(* Logix 5000 project; controller TBEN_Lx_8IOL_AOI_V0_1 vendor 1 type 14 code 176 rev 32.11; software revision 32.00; part 11 of 11 *)
(* tags used below, declared in another part *)
   Port : INT;
   Universal_IOLink_Info : Universal_IOLink_Info;
   StartupDone : BOOL;
   Done : DINT;
   Error : DINT;
   Active : DINT;
   Pending : DINT;
   Pending_or_Active : DINT;
   Status : DINT;
   ErrorCount : DINT;
   Prev_Vendor_ID : INT;
(* Universal_Device_Info, continued *)

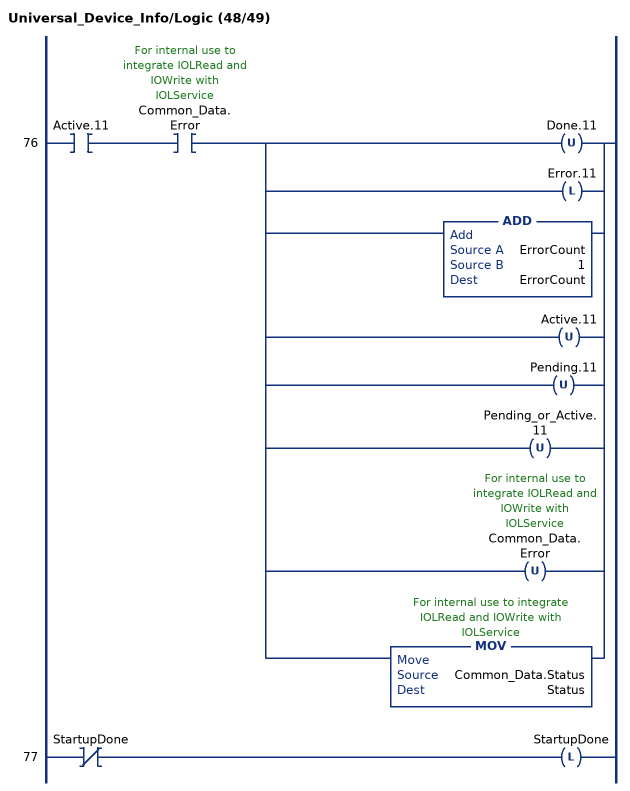
   [picture p96: Universal_Device_Info/Logic rungs 76-77]
   76: XIC(Active.11)XIC(Common_Data.Error)[OTU(Done.11) ,OTL(Error.11) ,ADD(ErrorCount,1,ErrorCount) ,OTU(Active.11) ,OTU(Pending.11) ,OTU(Pending_or_Active.11) ,OTU(Common_Data.Error) ,MOV(Common_Data.Status,Status) ];
   77: XIO(StartupDone)OTL(StartupDone);
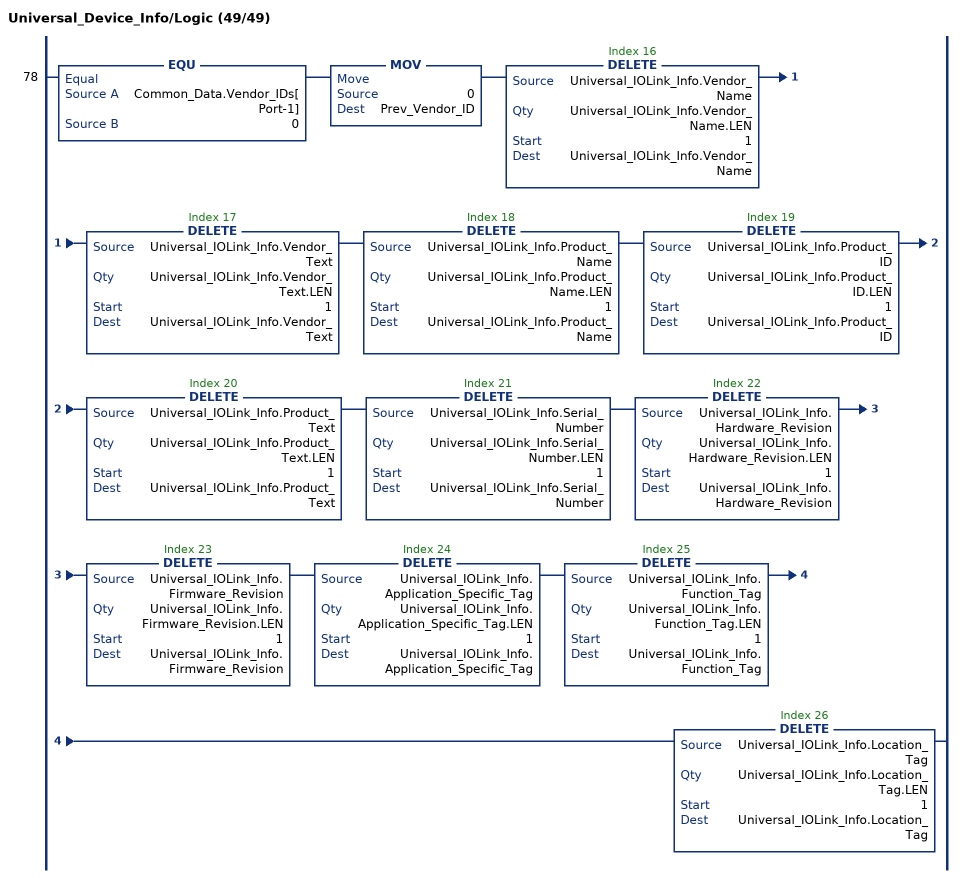
   78: EQU(Common_Data.Vendor_IDs[Port-1],0)MOV(0,Prev_Vendor_ID)DELETE(Universal_IOLink_Info.Vendor_Name,Universal_IOLink_Info.Vendor_Name.LEN,1,Universal_IOLink_Info.Vendor_Name)DELETE(Universal_IOLink_Info.Vendor_Text,Universal_IOLink_Info.Vendor_Text.LEN,1,Universal_IOLink_Info.Vendor_Text)DELETE(Universal_IOLink_Info.Product_Name,Universal_IOLink_Info.Product_Name.LEN,1,Universal_IOLink_Info.Product_Name)DELETE(Universal_IOLink_Info.Product_ID,Universal_IOLink_Info.Product_ID.LEN,1,Universal_IOLink_Info.Product_ID)DELETE(Universal_IOLink_Info.Product_Text,Universal_IOLink_Info.Product_Text.LEN,1,Universal_IOLink_Info.Product_Text)DELETE(Universal_IOLink_Info.Serial_Number,Universal_IOLink_Info.Serial_Number.LEN,1,Universal_IOLink_Info.Serial_Number)DELETE(Universal_IOLink_Info.Hardware_Revision,Universal_IOLink_Info.Hardware_Revision.LEN,1,Universal_IOLink_Info.Hardware_Revision)DELETE(Universal_IOLink_Info.Firmware_Revision,Universal_IOLink_Info.Firmware_Revision.LEN,1,Universal_IOLink_Info.Firmware_Revision)DELETE(Universal_IOLink_Info.Application_Specific_Tag,Universal_IOLink_Info.Application_Specific_Tag.LEN,1,Universal_IOLink_Info.Application_Specific_Tag)DELETE(Universal_IOLink_Info.Function_Tag,Universal_IOLink_Info.Function_Tag.LEN,1,Universal_IOLink_Info.Function_Tag)DELETE(Universal_IOLink_Info.Location_Tag,Universal_IOLink_Info.Location_Tag.LEN,1,Universal_IOLink_Info.Location_Tag);
END_ROUTINE

ROUTINE Prescan   (* ladder *)
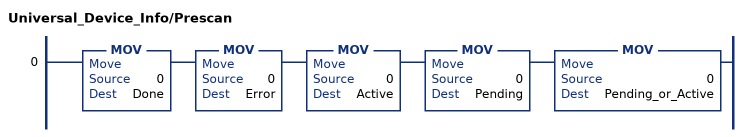
   0: MOV(0,Done)MOV(0,Error)MOV(0,Active)MOV(0,Pending)MOV(0,Pending_or_Active);
END_ROUTINE
END_ADD_ON_INSTRUCTION

VAR_GLOBAL   (* controller tags *)
   Common_Data : Turck_IOLink_Common_Data := (Port := 128, Index := -1, SubIndex := 68, Length := 224, NextTicketNum := 1, Process_Input_Data[0] := 192, ReceiveData[10] := 1, ReceiveData[11] := 61, ReceiveData[13] := 30, ReceiveData[14] := 51, ReceiveData[15] := 3, ReceiveData[18] := 48, ReceiveData[19] := 48, ReceiveData[20] := 48, ReceiveData[21] := 49, ReceiveData[22] := 48, ReceiveData[23] := 55, ReceiveData[24] := 54, ReceiveData[25] := 54, ReceiveData[26] := 53, ReceiveData[27] := 56, ReceiveData[28] := 45, ReceiveData[29] := 48, ReceiveData[30] := 48, ReceiveData[31] := 48, ReceiveData[32] := 50, ReceiveData[33] := 48, ReceiveData[34] := 17, ReceiveData[35] := 16, ReceiveData[36] := 16, ReceiveData[37] := 32, SendData[0] := -1, SendData[1] := -1, SendData[2] := 68, Vendor_IDs[0] := 317, Device_IDs[0] := 1979139);
   IOL_READ_MSG : MESSAGE;
        MessageParameters(ServiceCode := 16#004b, LocalElement := Common_Data.SendData, DestinationTag := Common_Data.ReceiveData, ...)
   IOL_WRITE_MSG : MESSAGE;
        MessageParameters(ServiceCode := 16#004c, LocalElement := Common_Data.SendData, DestinationTag := Common_Data.ReceiveData, ...)
   TBEN_8IOL_101 : TBEN_Lx_8IOL_AOI;
   TBEN_8IOL_101_Config_Tags_IN : Generic_160_SINT;
   TBEN_8IOL_101_Config_Tags_OUT : Generic_160_SINT;
   TBEN_8IOL_101_Process_Data_In : Generic_173_Words := (Data[0] := 1, Data[2] := 1, Data[3] := 192, Data[134] := 4, Data[135] := 4, Data[136] := 4, Data[137] := 4, Data[138] := 4, Data[139] := 4, Data[140] := 4);
   TBEN_8IOL_101_Process_Data_Out : Generic_131_Words;
   TBIL : Universal_Device_Info := (Port := 5);
   TBIL_Info : Universal_IOLink_Info;
   TEST : BOOL;
END_VAR

PROGRAM MainProgram   (* main routine MainRoutine *)
VAR
   TBEN_8IOL_100_Process_Data_In : Generic_173_Words := (Data[0] := 1, Data[133] := 4, Data[134] := 4, Data[135] := 4, Data[136] := 4, Data[137] := 4, Data[138] := 4, Data[139] := 4, Data[140] := 4);
   TBEN_8IOL_100_Process_Data_Out : Generic_131_Words;
END_VAR

ROUTINE MainRoutine   (* ladder *)
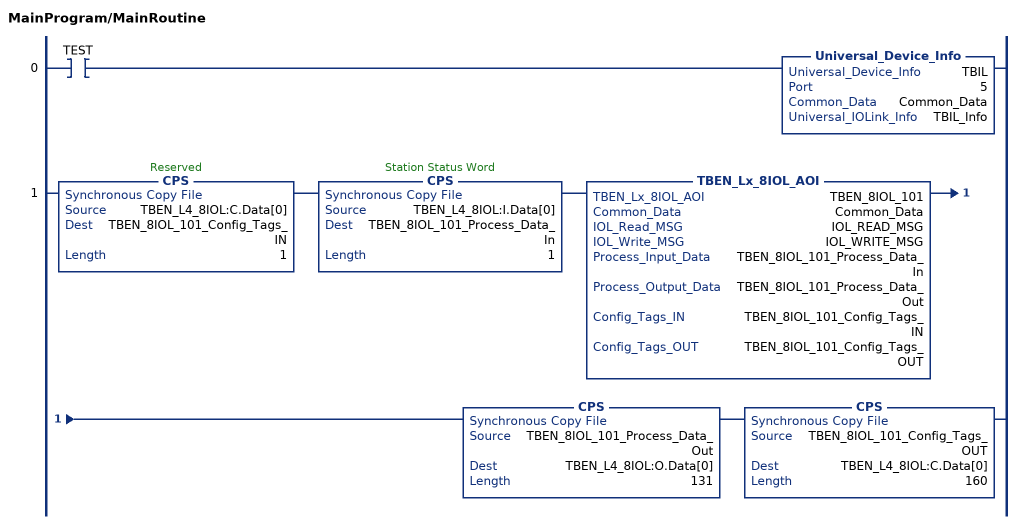
   0: XIC(TEST)Universal_Device_Info(TBIL,5,Common_Data,TBIL_Info);
   1: CPS(TBEN_L4_8IOL:C.Data[0],TBEN_8IOL_101_Config_Tags_IN,1)CPS(TBEN_L4_8IOL:I.Data[0],TBEN_8IOL_101_Process_Data_In,1)TBEN_Lx_8IOL_AOI(TBEN_8IOL_101,Common_Data,IOL_READ_MSG,IOL_WRITE_MSG,TBEN_8IOL_101_Process_Data_In,TBEN_8IOL_101_Process_Data_Out,TBEN_8IOL_101_Config_Tags_IN,TBEN_8IOL_101_Config_Tags_OUT)CPS(TBEN_8IOL_101_Process_Data_Out,TBEN_L4_8IOL:O.Data[0],131)CPS(TBEN_8IOL_101_Config_Tags_OUT,TBEN_L4_8IOL:C.Data[0],160);
END_ROUTINE
END_PROGRAM

PROGRAM SafetyProgram   (* main routine MainRoutine, safety *)

ROUTINE MainRoutine   (* ladder *)
END_ROUTINE
END_PROGRAM
